{attribute 'linkalways'} 
{attribute 'no_explicit_call' := 'This FB is a CLASS and must be accessed using methods or properties'}
{attribute 'enable_dynamic_creation'}
FUNCTION_BLOCK FINAL XOR_DINT EXTENDS Node
VAR
	in1 : _DINT(0);
	in2 : _DINT(0);
	out : _DINT(0);
END_VAR

METHOD PUBLIC Clone : I_Node
VAR
	pNode : POINTER TO XOR_DINT;
END_VAR
pNode := __NEW(XOR_DINT);
Clone := pNode^;
END_METHOD

METHOD FB_init : BOOL
VAR_INPUT
	bInitRetains : BOOL; // if TRUE, the retain variables are initialized (warm start / cold start)
	bInCopyCode : BOOL;  // if TRUE, the instance afterwards gets moved into the copy code (online change)
END_VAR
AddInput('in1',THIS^.in1);
AddInput('in2',THIS^.in2);
AddOutput('out', THIS^.out);
END_METHOD

METHOD PROTECTED OnExecute
VAR
END_VAR
out.Value := in1.Value XOR in2.Value;
END_METHOD

END_FUNCTION_BLOCK

(* stored: Version 1.1.0.1, ProductVersion 3.1.4024.15
   POU XOR_DINT: Id {e4a18d9a-c87d-42ed-9440-f861aa2c861c}, SpecialFunc None
   Folder Constructor: Id {18517766-2881-4249-b92d-527589669950}
   Method Clone: Id {3154f46c-6dba-412d-8e79-0ac8e8429132}
   Method FB_init: Id {cfcef46a-2008-4901-869f-5044e290d034}
   Method OnExecute: Id {c9ba5809-bc19-4004-95f7-a1823cb25346} *)
